// TIA Portal project "RFIDstuff" (V18)

(* hardware
DEVICE "S7-300/ET200M station_1"  S7-300 station
   slot 0: "Rail_0"  Rail  6ES7 390-1***0-0AA0
   slot 2: "PLC_1"  CPU 315-2 PN/DP  6ES7 315-2EH13-0AB0  V2.6
      slot 1: "MPI/DP interface_1"  X1
      slot 2: "PROFINET interface_1"  PN-IO
         slot 1: "Port_1"  Port
*)

// ===== PLC "PLC_1"  CPU 315-2 PN/DP =====

DATA_BLOCK "Data_block_2"   // DB5
{ S7_Optimized_Access := 'FALSE' }
VERSION : 0.1
   VAR
      greeting : String := 'PLC: hello world';
      testNumber : DInt := 8;
   END_VAR
BEGIN
END_DATA_BLOCK

DATA_BLOCK "Data_block_1"   // DB6
{ S7_Optimized_Access := 'FALSE' }
VERSION : 0.1
   VAR
      receivedData : String;
      disconnect : Bool;
      handshake : String := 'I am the PLC <|EOM|>';
      start : Bool;
      send : Bool := false;
      connected : Bool;
   END_VAR
BEGIN
END_DATA_BLOCK

ORGANIZATION_BLOCK "Main"   // OB1, LAD
TITLE = "Main Program Sweep (Cycle)"
{ S7_Optimized_Access := 'FALSE' }
VERSION : 0.1
   VAR_TEMP
      OB1_EV_CLASS : Byte;   // Bits 0-3 = 1 (Coming event), Bits 4-7 = 1 (Event class 1)
      OB1_SCAN_1 : Byte;   // 1 (Cold restart scan 1 of OB 1), 3 (Scan 2-n of OB 1)
      OB1_PRIORITY : Byte;   // Priority of OB Execution
      OB1_OB_NUMBR : Byte;   // 1 (Organization block 1, OB1)
      OB1_RESERVED_1 : Byte;   // Reserved for system
      OB1_RESERVED_2 : Byte;   // Reserved for system
      OB1_PREV_CYCLE : Int;   // Cycle time of previous OB1 scan (milliseconds)
      OB1_MIN_CYCLE : Int;   // Minimum cycle time of OB1 (milliseconds)
      OB1_MAX_CYCLE : Int;   // Maximum cycle time of OB1 (milliseconds)
      OB1_DATE_TIME : Date_And_Time;   // Date and time OB1 started
   END_VAR
BEGIN

REGION Network 1: Function to be executed on rising edge
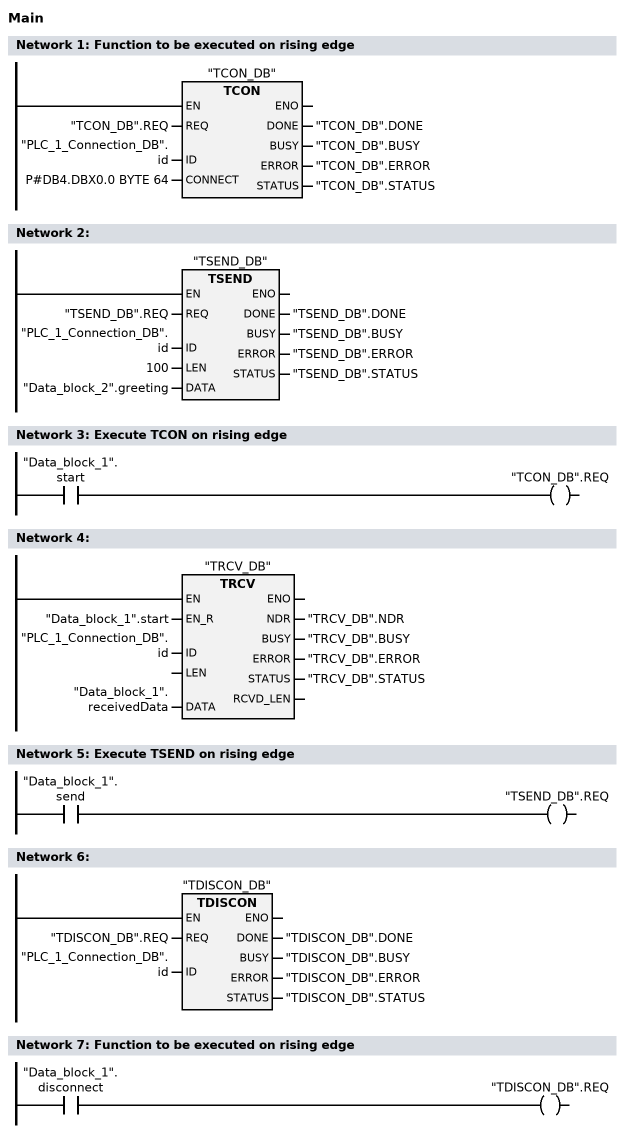
   "TCON_DB"(REQ := "TCON_DB".REQ,   // TCON
             ID := "PLC_1_Connection_DB".id,
             CONNECT := P#DB4.DBX0.0 BYTE 64,
             DONE => "TCON_DB".DONE,
             BUSY => "TCON_DB".BUSY,
             ERROR => "TCON_DB".ERROR,
             STATUS => "TCON_DB".STATUS);
END_REGION

REGION Network 2
   "TSEND_DB"(REQ := "TSEND_DB".REQ,   // TSEND
              ID := "PLC_1_Connection_DB".id,
              LEN := 100,
              DATA := "Data_block_2".greeting,
              DONE => "TSEND_DB".DONE,
              BUSY => "TSEND_DB".BUSY,
              ERROR => "TSEND_DB".ERROR,
              STATUS => "TSEND_DB".STATUS);
END_REGION

REGION Network 3: Execute TCON on rising edge
   RUNG wire#powerrail
      Contact( "Data_block_1".start )
      Coil( "TCON_DB".REQ )
   END_RUNG
   // the same network as SCL:
   "TCON_DB".REQ := "Data_block_1".start;
END_REGION

REGION Network 4
   "TRCV_DB"(EN_R := "Data_block_1".start,   // TRCV
             ID := "PLC_1_Connection_DB".id,
             DATA := "Data_block_1".receivedData,
             NDR => "TRCV_DB".NDR,
             BUSY => "TRCV_DB".BUSY,
             ERROR => "TRCV_DB".ERROR,
             STATUS => "TRCV_DB".STATUS);
END_REGION

REGION Network 5: Execute TSEND on rising edge
   RUNG wire#powerrail
      Contact( "Data_block_1".send )
      Coil( "TSEND_DB".REQ )
   END_RUNG
   // the same network as SCL:
   "TSEND_DB".REQ := "Data_block_1".send;
END_REGION

REGION Network 6
   "TDISCON_DB"(REQ := "TDISCON_DB".REQ,   // TDISCON
                ID := "PLC_1_Connection_DB".id,
                DONE => "TDISCON_DB".DONE,
                BUSY => "TDISCON_DB".BUSY,
                ERROR => "TDISCON_DB".ERROR,
                STATUS => "TDISCON_DB".STATUS);
END_REGION

REGION Network 7: Function to be executed on rising edge
   RUNG wire#powerrail
      Contact( "Data_block_1".disconnect )
      Coil( "TDISCON_DB".REQ )
   END_RUNG
   // the same network as SCL:
   "TDISCON_DB".REQ := "Data_block_1".disconnect;
END_REGION
END_ORGANIZATION_BLOCK